(* CODESYS project CodesysElevator.project

Project tree, tasks and I/O mapping:
  CODESYS_Control_Win_V3_x64 : CODESYS Control Win V3 x64, 3S - Smart Software Solutions GmbH, version 3.5.12.30
    application Application
      libraries: BASIC, 3.31 (OSCAT); Util, * (System)
      task VISU_TASK (cyclic, interval 50 ms, priority 31) calls VisuElems.Visu_Prg
      task Task (cyclic, interval t#20ms, priority 1) calls SimulationLogic, main
      Simulation/
        simcomponents/
          visualisation FloorButtons
          visualisation Door
          visualisation Elevator
        SimulationHelpers/
          function block MoveObject [ST]
          function block DoorLogic [ST]
        simlogic/
          program SimIO [ST]
          program SimulationLogic [ST]
        visualisation theLab
      IOs/
        global variables SystemState
        global variables IO
      control/
        program main [ST]
        function block last_floor_manager [LD]
        function block floor_request_handler [FBD]
        function block emergcy_handler [FBD]
        function block door_ctrl [SFC]
        program ElevatorControl [LD]
  libraries: SysTimeCore, 3.5.5.0 (System)
  text list GlobalTextList
*)

// CODESYS_Control_Win_V3_x64/Application/IOs/SystemState
VAR_GLOBAL
	useInputsFromSimulation: BOOL := TRUE;
END_VAR

// CODESYS_Control_Win_V3_x64/Application/IOs/IO
VAR_GLOBAL
	// inputs
	// Buttons
	ixButtonInElevatorF1: BOOL; // a request in the elevator to go to floor 1
	ixButtonInElevatorF2: BOOL;
	ixButtonInElevatorF3: BOOL;
	ixButtonInElevatorF4: BOOL;
	ixButtonInElevatorCloseDoors: BOOL; // a request to close the door inside the elevator if possible
	ixButtonInElevatorOpenDoors: BOOL; // a request to open the door inside the elevator if possible
	
	// security and sensors
	ixEmergencyStop: BOOL; // Emergency stop is pressed
	ixElevatorAt1: BOOL; // the elevator is at F1 sensor
	ixElevatorAt2: BOOL;
	ixElevatorAt3: BOOL;
	ixElevatorAt4: BOOL;
	ixDoorOpenedF1: BOOL; // the door is fully opened at F1
	ixDoorClosedF1: BOOL; // the door is fully closed at F1
	ixDoorOpenedF2: BOOL;
	ixDoorClosedF2: BOOL;
	ixDoorOpenedF3: BOOL;
	ixDoorClosedF3: BOOL;
	ixDoorOpenedF4: BOOL;
	ixDoorClosedF4: BOOL;

	// outputs
	// lamps
	qxLampInElevatorF1: BOOL;
	qxLampInElevatorF2: BOOL;
	qxLampInElevatorF3: BOOL;
	qxLampInElevatorF4: BOOL;
	qxLampEmergencyStop: BOOL;
	
	qxElevatorGoUp: BOOL;
	qxElevatorGoDown: BOOL;
	qxOpenDoorF1: BOOL; // Opens the door at F1, closes if false
	qxOpenDoorF2: BOOL; // Opens the door at F1, closes if false
	qxOpenDoorF3: BOOL; // Opens the door at F1, closes if false
	qxOpenDoorF4: BOOL; // Opens the door at F1, closes if false
	
END_VAR

// CODESYS_Control_Win_V3_x64/Application/Simulation/simlogic/SimulationLogic
PROGRAM SimulationLogic
VAR
	moveElevator: MoveObject;
	onlyForSimulationElevatorPosY: INT := 0;
	dummyZeroPos: INT := 0;
	elevatorMoving: BOOL;
	
	doorHandleF1: DoorLogic;
	leftPosF1: INT;
	rightPosF1: INT;	
	
	doorHandleF2: DoorLogic;
	leftPosF2: INT;
	rightPosF2: INT;	
	
	doorHandleF3: DoorLogic;
	leftPosF3: INT;
	rightPosF3: INT;	
	
	doorHandleF4: DoorLogic;
	leftPosF4: INT;
	rightPosF4: INT;
	

	
END_VAR


SimIO();



doorHandleF1(leftPos:=leftPosF1, rightPos:= rightPosF1, sensor:= ixElevatorAt1, open := qxOpenDoorF1, close := NOT qxOpenDoorF1);
doorHandleF2(leftPos:=leftPosF2, rightPos:= rightPosF2, sensor:= ixElevatorAt2, open := qxOpenDoorF2, close := NOT qxOpenDoorF2);
doorHandleF3(leftPos:=leftPosF3, rightPos:= rightPosF3, sensor:= ixElevatorAt3, open := qxOpenDoorF3, close := NOT qxOpenDoorF3);
doorHandleF4(leftPos:=leftPosF4, rightPos:= rightPosF4, sensor:= ixElevatorAt4, open := qxOpenDoorF4, close := NOT qxOpenDoorF4);
	

moveElevator(
	moveUP:= SimIO.sim_qxElevatorGoUp, 
	moveDown:= SimIO.sim_qxElevatorGoDown, 
	moveLeft:=FALSE , 
	moveRight:=FALSE , 
	maxX:=0, 
	minX:=0, 
	maxY:=340, 
	minY:=-30, 
	tick:=T#0.03S , 
	x:= dummyZeroPos, 
	y:= onlyForSimulationElevatorPosY );
	
elevatorMoving := moveElevator.isMoving;

END_PROGRAM

// CODESYS_Control_Win_V3_x64/Application/Simulation/simlogic/SimIO
PROGRAM SimIO
VAR
	
	simpleHysteresis: INT := 2;
	posF4: INT := -23;
	posF3: INT := 97;
	posF2: INT := 218;
	posF1: INT := 338;
	
		// for internal simulation use and a way to change bewteen sim and real
	sim_ixButtonAtF1Up: BOOL; 
	sim_ixButtonAtF2Down: BOOL; 
	sim_ixButtonAtF2Up: BOOL;   
	sim_ixButtonAtF3Down: BOOL;
	sim_ixButtonAtF3Up: BOOL;
	sim_ixButtonAtF4Down: BOOL;
	sim_ixButtonInElevatorF1: BOOL; 
	sim_ixButtonInElevatorF2: BOOL;
	sim_ixButtonInElevatorF3: BOOL;
	sim_ixButtonInElevatorF4: BOOL;
	sim_ixButtonInElevatorCloseDoors: BOOL; 
	sim_ixButtonInElevatorOpenDoors: BOOL; 
	
	sim_ixDoorSensorInElevator: BOOL; 
	sim_ixEmergencyStop: BOOL; 
	sim_ixElevatorAt1: BOOL; 
	sim_ixElevatorAt2: BOOL;
	sim_ixElevatorAt3: BOOL;
	sim_ixElevatorAt4: BOOL;
	sim_ixDoorOpenedF1: BOOL; 
	sim_ixDoorClosedF1: BOOL; 
	sim_ixDoorOpenedF2: BOOL;
	sim_ixDoorClosedF2: BOOL;
	sim_ixDoorOpenedF3: BOOL;
	sim_ixDoorClosedF3: BOOL;
	sim_ixDoorOpenedF4: BOOL;
	sim_ixDoorClosedF4: BOOL;

	sim_qxLampAtF1Up: BOOL;
	sim_qxLampAtF2Down: BOOL;
	sim_qxLampAtF2Up: BOOL;
	sim_qxLampAtF3Down: BOOL;
	sim_qxLampAtF3Up: BOOL;
	sim_qxLampAtF4Down: BOOL;
	sim_qxLampInElevatorF1: BOOL;
	sim_qxLampInElevatorF2: BOOL;
	sim_qxLampInElevatorF3: BOOL;
	sim_qxLampInElevatorF4: BOOL;
	sim_qxLampEmergencyStop: BOOL;
	
	sim_qxElevatorGoUp: BOOL;
	sim_qxElevatorGoDown: BOOL;
	sim_qxOpenDoorF1: BOOL; 
	sim_qxOpenDoorF2: BOOL; 
	sim_qxOpenDoorF3: BOOL; 
	sim_qxOpenDoorF4: BOOL; 
END_VAR

// logic

SimIO.sim_ixElevatorAt1 := SimulationLogic.onlyForSimulationElevatorPosY > posF1;
SimIO.sim_ixElevatorAt2 := SimulationLogic.onlyForSimulationElevatorPosY < posF2+simpleHysteresis AND SimulationLogic.onlyForSimulationElevatorPosY > posF2-simpleHysteresis;
SimIO.sim_ixElevatorAt3 := SimulationLogic.onlyForSimulationElevatorPosY < posF3+simpleHysteresis AND SimulationLogic.onlyForSimulationElevatorPosY > posF3-simpleHysteresis;
SimIO.sim_ixElevatorAt4 := SimulationLogic.onlyForSimulationElevatorPosY < posF4;

sim_ixDoorOpenedF1 := SimulationLogic.doorHandleF1.opened;
sim_ixDoorClosedF1 := SimulationLogic.doorHandleF1.closed;
sim_ixDoorOpenedF2 := SimulationLogic.doorHandleF2.opened;
sim_ixDoorClosedF2 := SimulationLogic.doorHandleF2.closed;
sim_ixDoorOpenedF3 := SimulationLogic.doorHandleF3.opened;
sim_ixDoorClosedF3 := SimulationLogic.doorHandleF3.closed;
sim_ixDoorOpenedF4 := SimulationLogic.doorHandleF4.opened;
sim_ixDoorClosedF4 := SimulationLogic.doorHandleF4.closed;


// mapping
IF useInputsFromSimulation THEN
	ixButtonInElevatorF1:=sim_ixButtonInElevatorF1;
	ixButtonInElevatorF2:=sim_ixButtonInElevatorF2;
	ixButtonInElevatorF3:=sim_ixButtonInElevatorF3;
	ixButtonInElevatorF4:=sim_ixButtonInElevatorF4;
	ixButtonInElevatorCloseDoors:=sim_ixButtonInElevatorCloseDoors;
	ixButtonInElevatorOpenDoors:=sim_ixButtonInElevatorOpenDoors;
	
	ixEmergencyStop:=sim_ixEmergencyStop;
	ixElevatorAt1:=sim_ixElevatorAt1;
	ixElevatorAt2:=sim_ixElevatorAt2;
	ixElevatorAt3:=sim_ixElevatorAt3;
	ixElevatorAt4:=sim_ixElevatorAt4;
	ixDoorOpenedF1:=sim_ixDoorOpenedF1;
	ixDoorClosedF1:=sim_ixDoorClosedF1;
	ixDoorOpenedF2:=sim_ixDoorOpenedF2;
	ixDoorClosedF2:=sim_ixDoorClosedF2;
	ixDoorOpenedF3:=sim_ixDoorOpenedF3;
	ixDoorClosedF3:=sim_ixDoorClosedF3;
	ixDoorOpenedF4:=sim_ixDoorOpenedF4;
	ixDoorClosedF4:=sim_ixDoorClosedF4;
END_IF

	sim_qxLampInElevatorF1:=qxLampInElevatorF1;
	sim_qxLampInElevatorF2:=qxLampInElevatorF2;
	sim_qxLampInElevatorF3:=qxLampInElevatorF3;
	sim_qxLampInElevatorF4:=qxLampInElevatorF4;
	sim_qxLampEmergencyStop:=qxLampEmergencyStop;
	
	sim_qxElevatorGoUp:=qxElevatorGoUp;
	sim_qxElevatorGoDown:=qxElevatorGoDown;
	sim_qxOpenDoorF1:=qxOpenDoorF1;
	sim_qxOpenDoorF2:=qxOpenDoorF2;
	sim_qxOpenDoorF3:=qxOpenDoorF3;
	sim_qxOpenDoorF4:=qxOpenDoorF4;

END_PROGRAM

// CODESYS_Control_Win_V3_x64/Application/Simulation/SimulationHelpers/MoveObject
FUNCTION_BLOCK MoveObject
VAR_INPUT
	moveUP: BOOL;
	moveDown: BOOL;
	moveLeft: BOOL;
	moveRight: BOOL;
	maxX: INT;
	minX: INT;
	maxY: INT;
	minY: INT;
	tick: time;
END_VAR
VAR_IN_OUT
	x: INT;
	y: INT;
END_VAR
VAR_OUTPUT
	isMoving: BOOL;
END_VAR
VAR
	pulse: CLK_PULSE;
END_VAR

pulse(
	PT:= tick, 
	N:= 0, 
	RST:= NOT moveUp AND NOT moveDown AND NOT moveLeft AND NOT moveRight , 
	Q=> , 
	CNT=> , 
	RUN=> );
	
IF pulse.Q THEN
	IF moveUP AND NOT moveDown AND y > minY THEN
		y := y-1; 
	ELSIF NOT moveUP AND moveDown AND y < maxY THEN
		y := y+1;
	END_IF
	
	IF moveRight AND NOT moveLeft AND x < maxX THEN
		x := x+1;
	ELSIF NOT moveRight AND moveLeft AND x > minX THEN
		x := x-1;
	END_IF
END_IF

isMoving := moveUP OR moveDown;

END_FUNCTION_BLOCK

// CODESYS_Control_Win_V3_x64/Application/Simulation/SimulationHelpers/DoorLogic
FUNCTION_BLOCK DoorLogic
VAR_INPUT
	open: BOOL;
	close: BOOL;
	sensor: BOOL;
END_VAR
VAR_OUTPUT
	opened: BOOL;
	closed: BOOL;
END_VAR
VAR_IN_OUT
	leftPos: INT;
	rightPos: INT;
END_VAR
VAR
	moveLeft: MoveObject;
	moveRight: MoveObject;
	dummy: INT;
	doOpen: BOOL;
	doClose: BOOL;
END_VAR


opened := leftPos <= -60 AND rightPos >= 60;
closed := leftPos >= 0 AND rightPos <= 0;

doOpen := open AND NOT opened AND NOT close;
doClose := close AND NOT closed AND NOT open;


moveLeft(
	moveUP:= FALSE, 
	moveDown:= FALSE, 
	moveLeft:=doOpen, 
	moveRight:=doClose, 
	maxX:=300, 
	minX:=-300, 
	maxY:=0, 
	minY:=0, 
	tick:=T#0.03S , 
	x:= leftPos, 
	y:= dummy
);

moveRight(
	moveUP:= FALSE, 
	moveDown:= FALSE, 
	moveLeft:=doClose , 
	moveRight:=doOpen , 
	maxX:=300, 
	minX:=-300, 
	maxY:=0, 
	minY:=0, 
	tick:=T#0.03S , 
	x:= rightPos, 
	y:= dummy
);

END_FUNCTION_BLOCK

// CODESYS_Control_Win_V3_x64/Application/control/main
PROGRAM main
VAR
END_VAR

ElevatorControl();

END_PROGRAM

// CODESYS_Control_Win_V3_x64/Application/control/ElevatorControl
PROGRAM ElevatorControl
VAR
	request1:BOOL;
	request2:BOOL;
	request3:BOOL;
	request4:BOOL :=TRUE;
	
	floor_request_handler:floor_request_handler;
	last_floor_manager:last_floor_manager;
	
	dorr_ctrl_1:door_ctrl;
	dorr_ctrl_2:door_ctrl;
	dorr_ctrl_3:door_ctrl;
	dorr_ctrl_4:door_ctrl;
	
	move_blocker:BOOL;
	emergency_blocker:BOOL;
	emergcy_handler:emergcy_handler;
END_VAR
VAR // added by the converter: edge detectors and wires of the graphical bodies
    _ft1, _ft2, _ft3, _ft4 : F_TRIG;
END_VAR

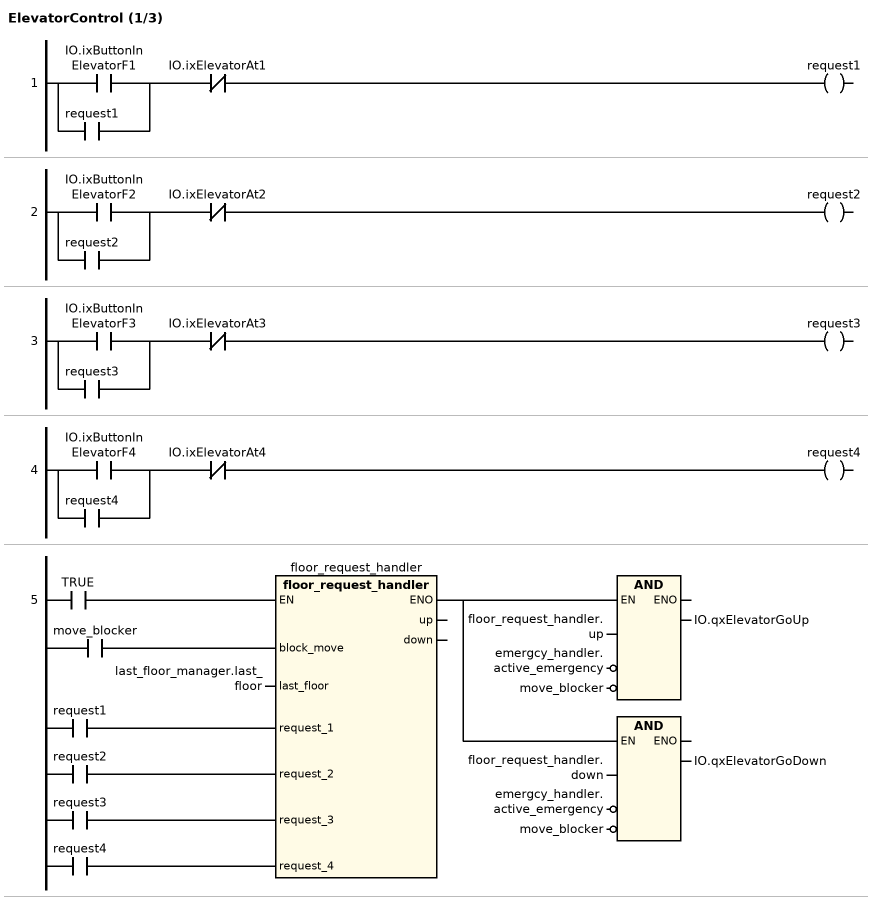
// NETWORK 1
request1 := (IO.ixButtonInElevatorF1 OR request1) AND NOT IO.ixElevatorAt1;

// NETWORK 2
request2 := (IO.ixButtonInElevatorF2 OR request2) AND NOT IO.ixElevatorAt2;

// NETWORK 3
request3 := (IO.ixButtonInElevatorF3 OR request3) AND NOT IO.ixElevatorAt3;

// NETWORK 4
request4 := (IO.ixButtonInElevatorF4 OR request4) AND NOT IO.ixElevatorAt4;

// NETWORK 5
floor_request_handler(
    block_move := move_blocker,
    last_floor := last_floor_manager.last_floor,
    request_1 := request1,
    request_2 := request2,
    request_3 := request3,
    request_4 := request4);
IO.qxElevatorGoUp := floor_request_handler.up AND NOT emergcy_handler.active_emergency AND NOT move_blocker;
IO.qxElevatorGoDown := floor_request_handler.down AND NOT emergcy_handler.active_emergency AND NOT move_blocker;

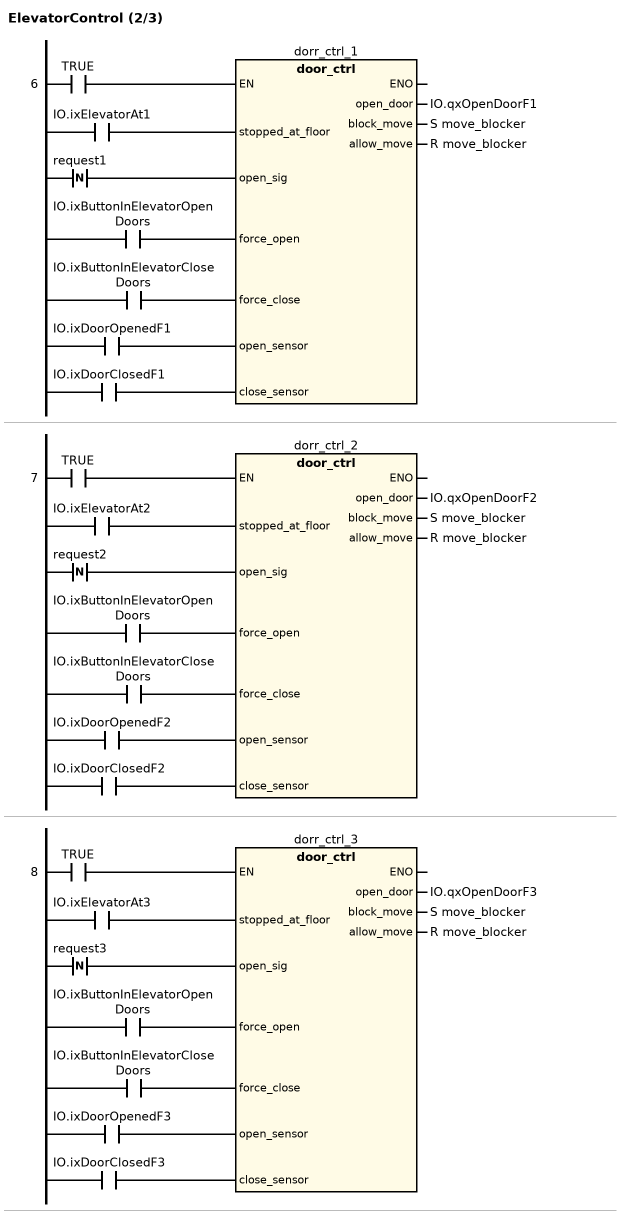
// NETWORK 6
_ft1(CLK := request1);
dorr_ctrl_1(
    stopped_at_floor := IO.ixElevatorAt1,
    open_sig := _ft1.Q,
    force_open := IO.ixButtonInElevatorOpenDoors,
    force_close := IO.ixButtonInElevatorCloseDoors,
    open_sensor := IO.ixDoorOpenedF1,
    close_sensor := IO.ixDoorClosedF1,
    open_door => IO.qxOpenDoorF1); // door_ctrl
move_blocker S= dorr_ctrl_1.block_move;
move_blocker R= dorr_ctrl_1.allow_move;

// NETWORK 7
_ft2(CLK := request2);
dorr_ctrl_2(
    stopped_at_floor := IO.ixElevatorAt2,
    open_sig := _ft2.Q,
    force_open := IO.ixButtonInElevatorOpenDoors,
    force_close := IO.ixButtonInElevatorCloseDoors,
    open_sensor := IO.ixDoorOpenedF2,
    close_sensor := IO.ixDoorClosedF2,
    open_door => IO.qxOpenDoorF2); // door_ctrl
move_blocker S= dorr_ctrl_2.block_move;
move_blocker R= dorr_ctrl_2.allow_move;

// NETWORK 8
_ft3(CLK := request3);
dorr_ctrl_3(
    stopped_at_floor := IO.ixElevatorAt3,
    open_sig := _ft3.Q,
    force_open := IO.ixButtonInElevatorOpenDoors,
    force_close := IO.ixButtonInElevatorCloseDoors,
    open_sensor := IO.ixDoorOpenedF3,
    close_sensor := IO.ixDoorClosedF3,
    open_door => IO.qxOpenDoorF3); // door_ctrl
move_blocker S= dorr_ctrl_3.block_move;
move_blocker R= dorr_ctrl_3.allow_move;

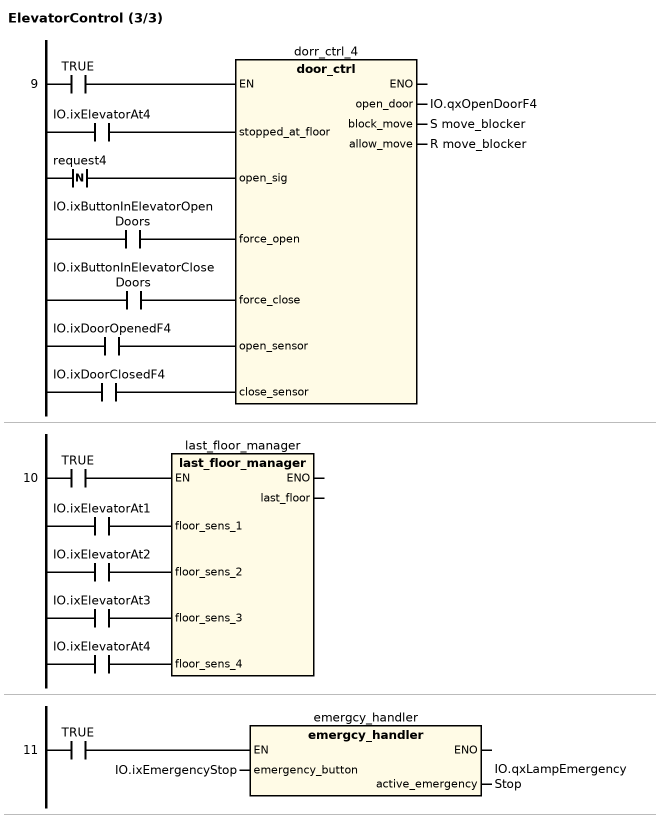
// NETWORK 9
_ft4(CLK := request4);
dorr_ctrl_4(
    stopped_at_floor := IO.ixElevatorAt4,
    open_sig := _ft4.Q,
    force_open := IO.ixButtonInElevatorOpenDoors,
    force_close := IO.ixButtonInElevatorCloseDoors,
    open_sensor := IO.ixDoorOpenedF4,
    close_sensor := IO.ixDoorClosedF4,
    open_door => IO.qxOpenDoorF4); // door_ctrl
move_blocker S= dorr_ctrl_4.block_move;
move_blocker R= dorr_ctrl_4.allow_move;

// NETWORK 10
last_floor_manager(
    floor_sens_1 := IO.ixElevatorAt1,
    floor_sens_2 := IO.ixElevatorAt2,
    floor_sens_3 := IO.ixElevatorAt3,
    floor_sens_4 := IO.ixElevatorAt4);

// NETWORK 11
emergcy_handler(emergency_button := IO.ixEmergencyStop, active_emergency => IO.qxLampEmergencyStop);

END_PROGRAM

// CODESYS_Control_Win_V3_x64/Application/control/floor_request_handler
FUNCTION_BLOCK floor_request_handler
VAR_INPUT
	block_move: BOOL;
	last_floor:INT;
	request_1:BOOL;
	request_2:BOOL;
	request_3:BOOL;
	request_4:BOOL;
	
END_VAR
VAR_OUTPUT
	up:BOOL;
	down:BOOL;
END_VAR
VAR
	floor1: INT:=1;
	floor2: INT:=2;
	floor3: INT:=3;
	floor4: INT:=4;
END_VAR

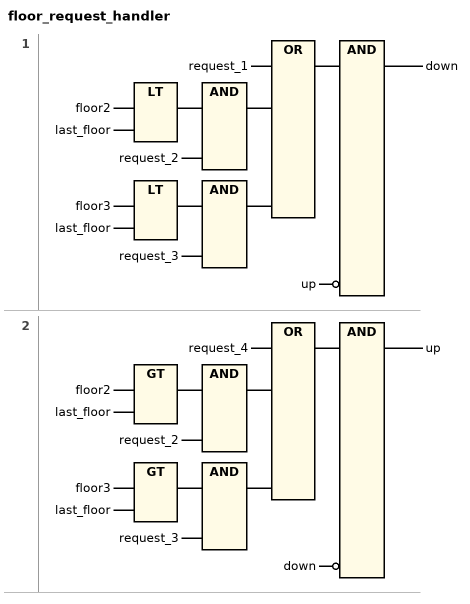
// NETWORK 1
down := (request_1 OR floor2 < last_floor AND request_2 OR floor3 < last_floor AND request_3) AND NOT up;

// NETWORK 2
up := (request_4 OR floor2 > last_floor AND request_2 OR floor3 > last_floor AND request_3) AND NOT down;

END_FUNCTION_BLOCK

// CODESYS_Control_Win_V3_x64/Application/control/last_floor_manager
FUNCTION_BLOCK last_floor_manager
VAR_INPUT
	floor_sens_1:BOOL;
	floor_sens_2:BOOL;
	floor_sens_3:BOOL;
	floor_sens_4:BOOL;
END_VAR
VAR_OUTPUT
	last_floor: INT := 4;
END_VAR
VAR
END_VAR
VAR // added by the converter: edge detectors and wires of the graphical bodies
    _rt1, _rt2, _rt3, _rt4 : R_TRIG;
END_VAR

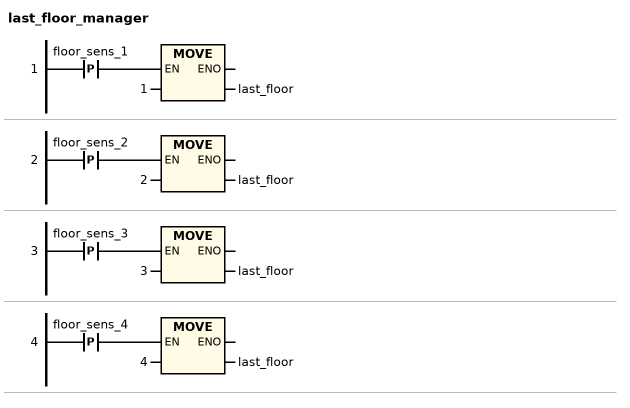
// NETWORK 1
_rt1(CLK := floor_sens_1);
IF _rt1.Q THEN last_floor := 1; END_IF

// NETWORK 2
_rt2(CLK := floor_sens_2);
IF _rt2.Q THEN last_floor := 2; END_IF

// NETWORK 3
_rt3(CLK := floor_sens_3);
IF _rt3.Q THEN last_floor := 3; END_IF

// NETWORK 4
_rt4(CLK := floor_sens_4);
IF _rt4.Q THEN last_floor := 4; END_IF

END_FUNCTION_BLOCK

// CODESYS_Control_Win_V3_x64/Application/control/emergcy_handler
FUNCTION_BLOCK emergcy_handler
VAR_INPUT
	emergency_button:BOOL;
END_VAR
VAR_OUTPUT
	active_emergency: BOOL;
END_VAR
VAR
	timer : TON;
	
END_VAR
VAR // added by the converter: edge detectors and wires of the graphical bodies
    _rt1 : R_TRIG;
END_VAR

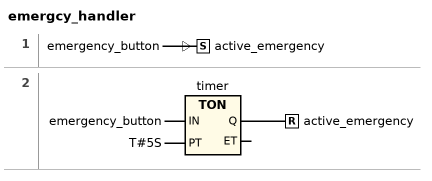
// NETWORK 1
_rt1(CLK := emergency_button);
active_emergency S= _rt1.Q;

// NETWORK 2
timer(IN := emergency_button, PT := T#5S); // TON
active_emergency R= timer.Q;

END_FUNCTION_BLOCK

// CODESYS_Control_Win_V3_x64/Application/control/door_ctrl
FUNCTION_BLOCK door_ctrl
VAR_INPUT
	stopped_at_floor:BOOL;
	open_sig:BOOL;
	force_open:BOOL;
	force_close:BOOL;
	open_sensor:BOOL;
	close_sensor:BOOL;
END_VAR
VAR_OUTPUT
	open_door:BOOL;
	block_move:BOOL;
	allow_move:BOOL;
END_VAR
VAR
END_VAR

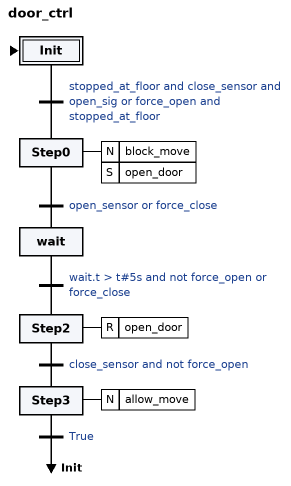
INITIAL_STEP Init:
END_STEP
TRANSITION FROM Init TO Step0
    := stopped_at_floor and close_sensor and open_sig or force_open and stopped_at_floor;
END_TRANSITION
STEP Step0:
    block_move(N);
    open_door(S);
END_STEP
TRANSITION FROM Step0 TO wait
    := open_sensor or force_close;
END_TRANSITION
STEP wait:
END_STEP
TRANSITION FROM wait TO Step2
    := wait.t > t#5s and not force_open or force_close;
END_TRANSITION
STEP Step2:
    open_door(R);
END_STEP
TRANSITION FROM Step2 TO Step3
    := close_sensor and not force_open;
END_TRANSITION
STEP Step3:
    allow_move(N);
END_STEP
TRANSITION FROM Step3 TO Init
    := True;
END_TRANSITION

END_FUNCTION_BLOCK

// CODESYS_Control_Win_V3_x64/Application/Simulation/simcomponents/FloorButtons
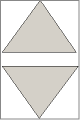
VISUALIZATION FloorButtons  // 80x120
VAR_IN_OUT
	clickUp: BOOL;
	clickDown: BOOL;
	lampUP: BOOL;
	lampDown: BOOL;
END_VAR
    Polygon (2,52) (40,0) (76,52), colour toggle: lampUP
        tap clickUp
    Polygon (2,66) (39,118) (78,66), colour toggle: lampDown
        tap clickDown
END_VISUALIZATION

// CODESYS_Control_Win_V3_x64/Application/Simulation/simcomponents/Door
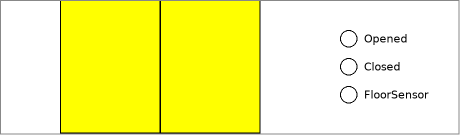
VISUALIZATION Door  // 460x135
VAR_IN_OUT
	opened: BOOL;
	closed: BOOL;
	sensor: BOOL;
	posL: INT;
	posR: INT;
END_VAR
    Rectangle (60,0 100x133)
        p3560616238: posL
    Rectangle (160,0 100x133)
        p3560616238: posR
    Ellipse (340,30 17x17), colour toggle: opened
    Label (361,24 57x30), "Opened"
    Ellipse (340,58 17x17), colour toggle: closed
    Label (361,52 57x30), "Closed"
    Ellipse (340,86 17x17), colour toggle: sensor
    Label (361,80 97x30), "FloorSensor"
END_VISUALIZATION

// CODESYS_Control_Win_V3_x64/Application/Simulation/theLab
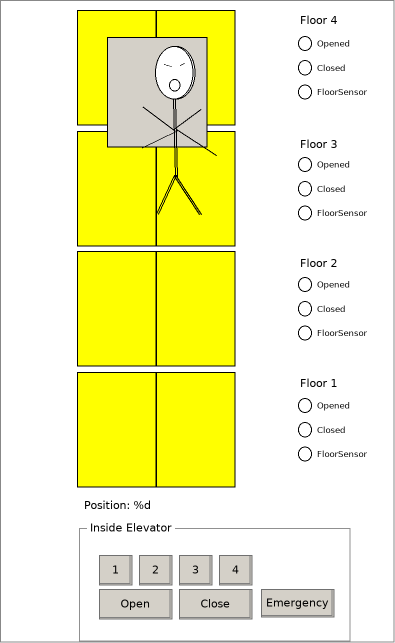
VISUALIZATION theLab  // 395x643
    Frame (30,372 363x117)
        shows Door(opened := SimulationLogic.doorHandleF1.opened, closed := SimulationLogic.doorHandleF1.closed, sensor := SimulationLogic.doorHandleF1.sensor, posL := SimulationLogic.leftPosF1, posR := SimulationLogic.rightPosF1)
    Frame (30,131 363x117)
        shows Door(opened := SimulationLogic.doorHandleF3.opened, closed := SimulationLogic.doorHandleF3.closed, sensor := SimulationLogic.doorHandleF3.sensor, posL := SimulationLogic.leftPosF3, posR := SimulationLogic.rightPosF3)
    Frame (30,251 363x117)
        shows Door(opened := SimulationLogic.doorHandleF2.opened, closed := SimulationLogic.doorHandleF2.closed, sensor := SimulationLogic.doorHandleF2.sensor, posL := SimulationLogic.leftPosF2, posR := SimulationLogic.rightPosF2)
    Frame (30,10 363x117)
        shows Door(opened := SimulationLogic.doorHandleF4.opened, closed := SimulationLogic.doorHandleF4.closed, sensor := SimulationLogic.doorHandleF4.sensor, posL := SimulationLogic.leftPosF4, posR := SimulationLogic.rightPosF4)
    Rectangle (81,494 179x23), "Position: %d", text variable: simulationLogic.onlyForSimulationElevatorPosY
    RoundedRectangle (107,37 100x110)
        p2738717112: SimulationLogic.onlyForSimulationElevatorPosY
    Group (142,46 38x95), invisible if: SimulationLogic.moveElevator.isMoving
        p2738717112: SimulationLogic.onlyForSimulationElevatorPosY
        Ellipse (15,0 38x53)
        Line (61,63)
        Line (33,53) (35,131)
        Line (34,83) (74,109)
        Line (35,85) (0,102)
        Line (34,129) (16,168)
        Line (34,130) (59,168)
        Line (26,39) (43,39)
        Line (23,24) (31,20)
        Line (40,19) (44,23)
    Group (143,46 31x95), invisible if: not SimulationLogic.elevatorMoving
        p2738717112: SimulationLogic.onlyForSimulationElevatorPosY
        Ellipse (12,0 38x53)
        Line (58,63)
        Line (30,53) (32,131)
        Line (31,83) (58,63)
        Line (32,85) (0,61)
        Line (31,129) (13,168)
        Line (31,130) (56,168)
        Line (21,18) (28,20)
        Line (37,19) (41,17)
        Ellipse (26,33 11x12)
    GroupBox (79,520 271x121), "Inside Elevator"
        Button (60,35 33x30), "2", colour toggle: SimIO.sim_qxLampInElevatorF2
            tap SimIO.sim_ixButtonInElevatorF2
        Button (100,35 33x30), "3", colour toggle: SimIO.sim_qxLampInElevatorF3
            tap SimIO.sim_ixButtonInElevatorF3
        Button (140,35 33x30), "4", colour toggle: SimIO.sim_qxLampInElevatorF4
            tap SimIO.sim_ixButtonInElevatorF4
        Button (20,35 33x30), "1", colour toggle: SimIO.sim_qxLampInElevatorF1
            tap SimIO.sim_ixButtonInElevatorF1
        Button (20,69 73x30), "Open"
            tap SimIO.sim_ixButtonInElevatorOpenDoors
        Button (100,69 73x30), "Close"
            tap SimIO.sim_ixButtonInElevatorCloseDoors
        Button (182,69 73x28), "Emergency"
            tap SimIO.sim_ixEmergencyStop
    Rectangle (297,372 56x23), "Floor 1"
    Rectangle (297,252 56x23), "Floor 2"
    Rectangle (297,133 56x23), "Floor 3"
    Rectangle (297,9 56x23), "Floor 4"
END_VISUALIZATION

// CODESYS_Control_Win_V3_x64/Application/Simulation/simcomponents/Elevator
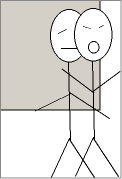
VISUALIZATION Elevator  // 122x179
VAR_IN_OUT
	moving: BOOL;
END_VAR
    RoundedRectangle (0,0 100x110), colour toggle: moving
    Group (35,9 38x95), invisible if: SimulationLogic.moveElevator.isMoving
        Ellipse (15,0 38x53)
        Line (61,63)
        Line (33,53) (35,131)
        Line (34,83) (74,109)
        Line (35,85) (0,102)
        Line (34,129) (16,168)
        Line (34,130) (59,168)
        Line (26,39) (43,39)
        Line (23,24) (31,20)
        Line (40,19) (44,23)
    Group (62,8 31x95), invisible if: not SimulationLogic.elevatorMoving
        Ellipse (12,0 38x53)
        Line (58,63)
        Line (30,53) (32,131)
        Line (31,83) (58,63)
        Line (32,85) (0,61)
        Line (31,129) (13,168)
        Line (31,130) (56,168)
        Line (21,18) (28,20)
        Line (37,19) (41,17)
        Ellipse (26,33 11x12)
END_VISUALIZATION
